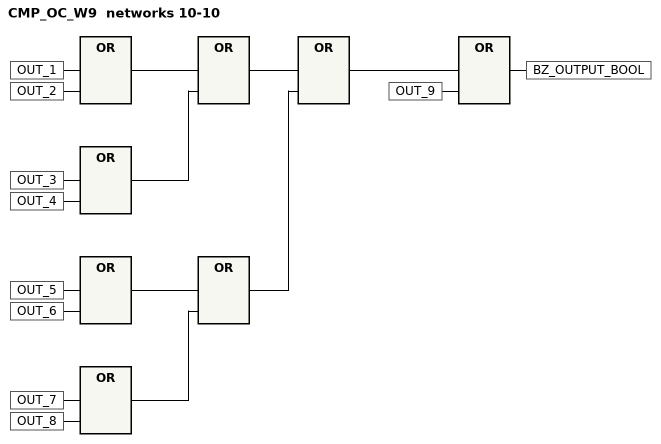
[picture p24: CMP_OC_W9 (FBD) networks 10-10]
_FBD_ (* Function Block Diagram *)
NETWORK 1
	OR(LT(WORD_1, 0), GT(WORD_1, 0)) => OUT_1
NETWORK 2
	OR(LT(WORD_2, 0), GT(WORD_2, 0)) => OUT_2
NETWORK 3
	OR(LT(WORD_3, 0), GT(WORD_3, 0)) => OUT_3
NETWORK 4
	OR(LT(WORD_4, 0), GT(WORD_4, 0)) => OUT_4
NETWORK 5
	OR(LT(WORD_5, 0), GT(WORD_5, 0)) => OUT_5
NETWORK 6
	OR(LT(WORD_6, 0), GT(WORD_6, 0)) => OUT_6
NETWORK 7
	OR(LT(WORD_7, 0), GT(WORD_7, 0)) => OUT_7
NETWORK 8
	OR(LT(WORD_8, 0), GT(WORD_8, 0)) => OUT_8
NETWORK 9
	OR(LT(WORD_9, 0), GT(WORD_9, 0)) => OUT_9
NETWORK 10
	OR(OR(OR(OR(OUT_1, OUT_2), OR(OUT_3, OUT_4)), OR(OR(OUT_5, OUT_6), OR(OUT_7, OUT_8))), OUT_9) => BZ_OUTPUT_BOOL
_END_FBD_
(* the same logic as Structured Text *)
(* Network 1 *)
OUT_1 := (WORD_1 < 0) OR (WORD_1 > 0);
(* Network 2 *)
OUT_2 := (WORD_2 < 0) OR (WORD_2 > 0);
(* Network 3 *)
OUT_3 := (WORD_3 < 0) OR (WORD_3 > 0);
(* Network 4 *)
OUT_4 := (WORD_4 < 0) OR (WORD_4 > 0);
(* Network 5 *)
OUT_5 := (WORD_5 < 0) OR (WORD_5 > 0);
(* Network 6 *)
OUT_6 := (WORD_6 < 0) OR (WORD_6 > 0);
(* Network 7 *)
OUT_7 := (WORD_7 < 0) OR (WORD_7 > 0);
(* Network 8 *)
OUT_8 := (WORD_8 < 0) OR (WORD_8 > 0);
(* Network 9 *)
OUT_9 := (WORD_9 < 0) OR (WORD_9 > 0);
(* Network 10 *)
BZ_OUTPUT_BOOL := (((OUT_1 OR OUT_2) OR (OUT_3 OR OUT_4)) OR ((OUT_5 OR OUT_6) OR (OUT_7 OR OUT_8))) OR OUT_9;
END_FUNCTION_BLOCK

(* POU DOWN_COUNT_TIMER, LD *)
FUNCTIONBLOCK DOWN_COUNT_TIMER
VAR_INPUT
	BOOL_SIGNAL_IN: BOOL;
	BOOL_TIMER_RST: BOOL;
	INT_AUTO_RST: INT;
	INT_SV_SEC: INT;
END_VAR
VAR_OUTPUT
	SIGNAL_BOOL: BOOL;
	PV_SEC_INT: INT;
END_VAR
VAR
	DF_1: R_TRIG;
	DF_2: R_TRIG;
	M1: BOOL;
	M2: BOOL;

	T100: TON;
	T101: TON;
	M100: BOOL;
	M101: BOOL;
	M200: BOOL;

	M110: BOOL;
	M300: BOOL;
END_VAR
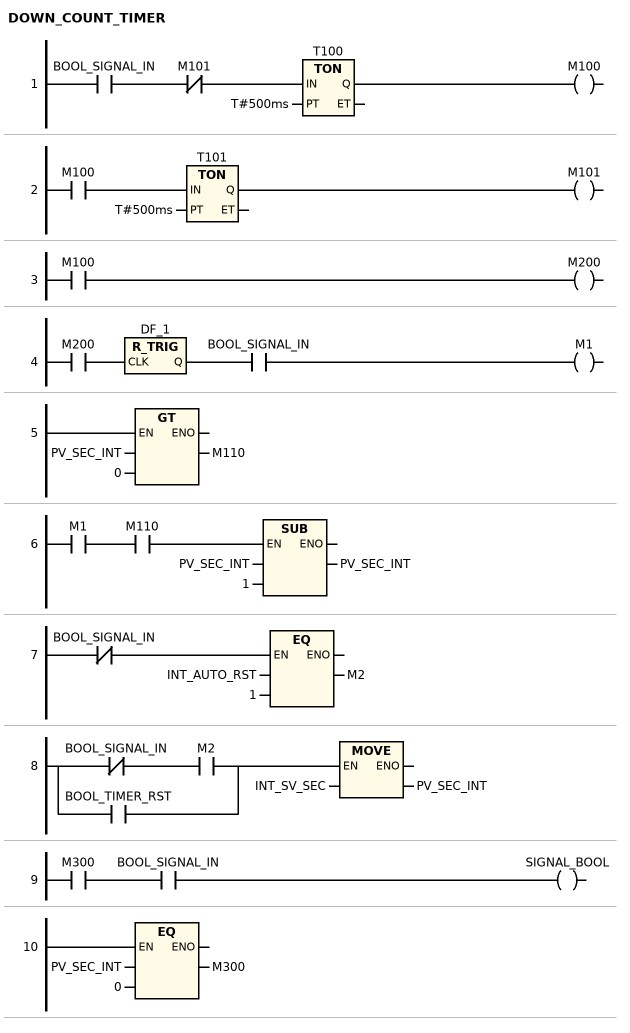
_LD_ (* Ladder Diagram *)
NETWORK 1
	[BOOL_SIGNAL_IN] - [/M101] - T100:TON(IN: *, PT: T#500ms) --- (M100)
NETWORK 2
	[M100] - T101:TON(IN: *, PT: T#500ms) --- (M101)
NETWORK 3
	[M100] --- (M200)
NETWORK 4
	[M200] - DF_1:R_TRIG(CLK: *) - [BOOL_SIGNAL_IN] --- (M1)
NETWORK 5
	*
		EN --- GT(PV_SEC_INT, 0) => M110
NETWORK 6
	[M1] - [M110]
		EN --- SUB(PV_SEC_INT, 1) => PV_SEC_INT
NETWORK 7
	[/BOOL_SIGNAL_IN]
		EN --- EQ(INT_AUTO_RST, 1) => M2
NETWORK 8
	{ [/BOOL_SIGNAL_IN] - [M2] | [BOOL_TIMER_RST] }
		EN --- MOVE(INT_SV_SEC) => PV_SEC_INT
NETWORK 9
	[M300] - [BOOL_SIGNAL_IN] --- (SIGNAL_BOOL)
NETWORK 10
	*
		EN --- EQ(PV_SEC_INT, 0) => M300
_END_LD_
(* the same logic as Structured Text *)
(* Network 1 *)
T100(IN := BOOL_SIGNAL_IN AND NOT M101, PT := T#500ms);
M100 := T100.Q;
(* Network 2 *)
T101(IN := M100, PT := T#500ms);
M101 := T101.Q;
(* Network 3 *)
M200 := M100;
(* Network 4 *)
DF_1(CLK := M200);
M1 := DF_1.Q AND BOOL_SIGNAL_IN;
(* Network 5 *)
M110 := PV_SEC_INT > 0;
(* Network 6 *)
IF M1 AND M110 THEN
	PV_SEC_INT := PV_SEC_INT - 1;
END_IF;
(* Network 7 *)
IF NOT BOOL_SIGNAL_IN THEN
	M2 := INT_AUTO_RST = 1;
END_IF;
(* Network 8 *)
IF NOT BOOL_SIGNAL_IN AND M2 OR BOOL_TIMER_RST THEN
	PV_SEC_INT := INT_SV_SEC;
END_IF;
(* Network 9 *)
SIGNAL_BOOL := M300 AND BOOL_SIGNAL_IN;
(* Network 10 *)
M300 := PV_SEC_INT = 0;
END_FUNCTION_BLOCK

(* POU CLOCK_PLS, LD *)
FUNCTION_BLOCK CLOCK_PLS
VAR_INPUT
	INT_TIME_ms : INT;

END_VAR
VAR_OUTPUT
	CLOCK_PLS_BOOL: BOOL;
END_VAR
VAR
	T0: TON;
	T1: TON;
	M0: BOOL;
	M1: BOOL;
	D0: TIME;
	D1: TIME;
END_VAR
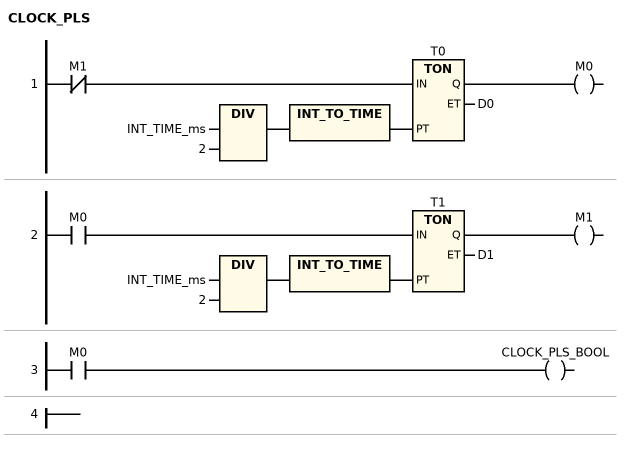
_LD_ (* Ladder Diagram *)
NETWORK 1
	[/M1] - T0:TON(IN: *, PT: INT_TO_TIME(DIV(INT_TIME_ms, 2)), ET => D0) --- (M0)
NETWORK 2
	[M0] - T1:TON(IN: *, PT: INT_TO_TIME(DIV(INT_TIME_ms, 2)), ET => D1) --- (M1)
NETWORK 3
	[M0] --- (CLOCK_PLS_BOOL)
NETWORK 4
	*
_END_LD_
(* the same logic as Structured Text *)
(* Network 1 *)
T0(IN := NOT M1, PT := INT_TO_TIME(INT_TIME_ms / 2));
D0 := T0.ET;
M0 := T0.Q;
(* Network 2 *)
T1(IN := M0, PT := INT_TO_TIME(INT_TIME_ms / 2));
D1 := T1.ET;
M1 := T1.Q;
(* Network 3 *)
CLOCK_PLS_BOOL := M0;
(* Network 4 *)
END_FUNCTION_BLOCK

(* POU EQ_GT, LD *)
FUNCTION_BLOCK EQ_GT
VAR_INPUT
	INT_SOURCE_A: INT;
	INT_SOURCE_B: INT;
END_VAR
VAR_OUTPUT
	SIGNAL_BOOL: BOOL;
END_VAR
VAR
	M0: BOOL;
	M1: BOOL;
END_VAR
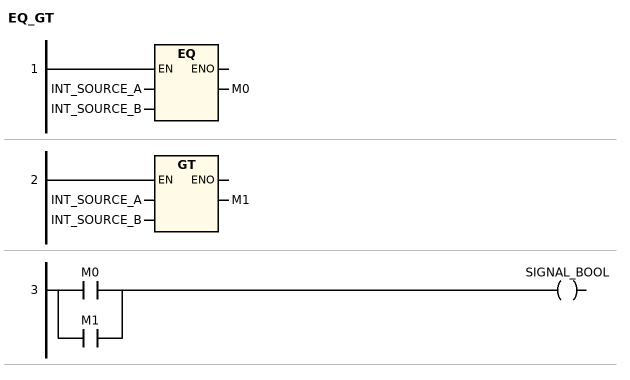
_LD_ (* Ladder Diagram *)
NETWORK 1
	*
		EN --- EQ(INT_SOURCE_A, INT_SOURCE_B) => M0
NETWORK 2
	*
		EN --- GT(INT_SOURCE_A, INT_SOURCE_B) => M1
NETWORK 3
	{ [M0] | [M1] } --- (SIGNAL_BOOL)
_END_LD_
(* the same logic as Structured Text *)
(* Network 1 *)
M0 := INT_SOURCE_A = INT_SOURCE_B;
(* Network 2 *)
M1 := INT_SOURCE_A > INT_SOURCE_B;
(* Network 3 *)
SIGNAL_BOOL := M0 OR M1;
END_FUNCTION_BLOCK

(* POU EQ_LT, LD *)
FUNCTION_BLOCK EQ_LT
VAR_INPUT
	INT_SOURCE_A:INT;
	INT_SOURCE_B:INT;
END_VAR
VAR_OUTPUT
	SIGNAL_BOOL:BOOL;
END_VAR
VAR
	M0: BOOL;
	M1: BOOL;
END_VAR
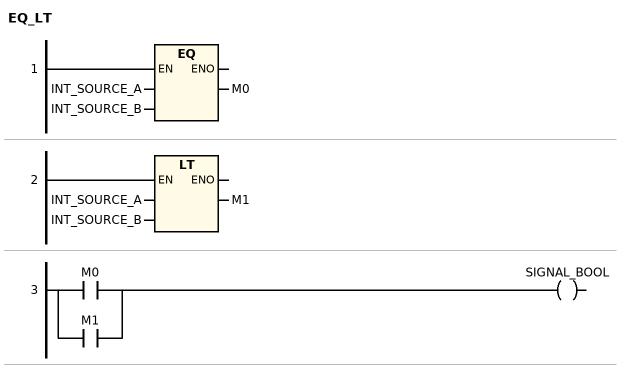
_LD_ (* Ladder Diagram *)
NETWORK 1
	*
		EN --- EQ(INT_SOURCE_A, INT_SOURCE_B) => M0
NETWORK 2
	*
		EN --- LT(INT_SOURCE_A, INT_SOURCE_B) => M1
NETWORK 3
	{ [M0] | [M1] } --- (SIGNAL_BOOL)
_END_LD_
(* the same logic as Structured Text *)
(* Network 1 *)
M0 := INT_SOURCE_A = INT_SOURCE_B;
(* Network 2 *)
M1 := INT_SOURCE_A < INT_SOURCE_B;
(* Network 3 *)
SIGNAL_BOOL := M0 OR M1;
END_FUNCTION_BLOCK

(* POU LT_GT, LD *)
FUNCTION_BLOCK LT_GT
VAR_INPUT
	INT_SOURCE_A: INT;
	INT_SOURCE_B: INT;
END_VAR
VAR_OUTPUT
	SIGNAL_BOOL: BOOL;
END_VAR
VAR
	M0: BOOL;
	M1: BOOL;
END_VAR
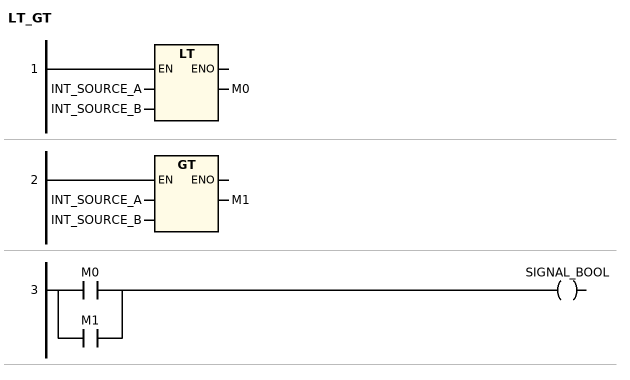
_LD_ (* Ladder Diagram *)
NETWORK 1
	*
		EN --- LT(INT_SOURCE_A, INT_SOURCE_B) => M0
NETWORK 2
	*
		EN --- GT(INT_SOURCE_A, INT_SOURCE_B) => M1
NETWORK 3
	{ [M0] | [M1] } --- (SIGNAL_BOOL)
_END_LD_
(* the same logic as Structured Text *)
(* Network 1 *)
M0 := INT_SOURCE_A < INT_SOURCE_B;
(* Network 2 *)
M1 := INT_SOURCE_A > INT_SOURCE_B;
(* Network 3 *)
SIGNAL_BOOL := M0 OR M1;
END_FUNCTION_BLOCK

(* POU TIMER_ALARM, LD *)
FUNCTION_BLOCK TIMER_ALARM
VAR_INPUT
	BOOL_SIGNAL_IN: BOOL;
	BOOL_ALMRST_PB: BOOL;
	BOOL_BZRST_PB: BOOL;
	INT_PV: INT;

END_VAR

VAR_OUTPUT
	ALM_MSG_BOOL: BOOL;
	BZ_OUT_BOOL: BOOL;
	EV_INT: INT;
END_VAR

VAR
	T1: TON;
	M0: BOOL;
	M1: BOOL;
	D200: TIME;
	D202: INT;
END_VAR
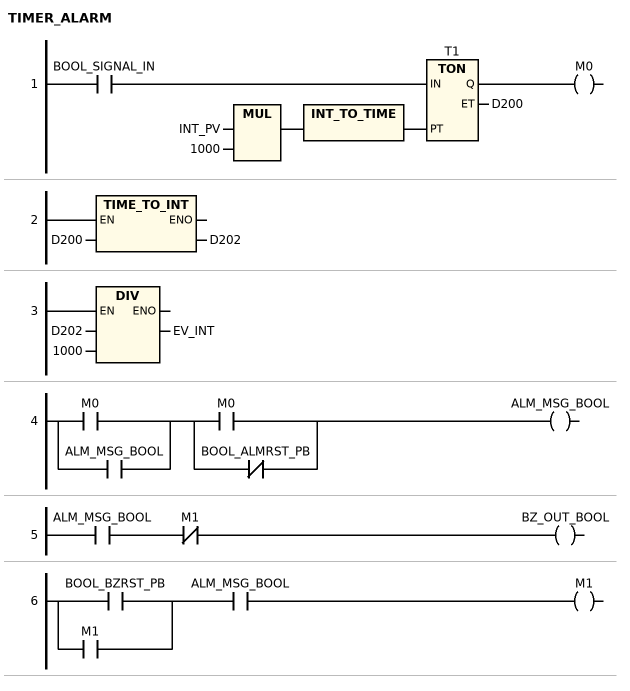
_LD_ (* Ladder Diagram *)
NETWORK 1
	[BOOL_SIGNAL_IN] - T1:TON(IN: *, PT: INT_TO_TIME(MUL(INT_PV, 1000)), ET => D200) --- (M0)
NETWORK 2
	*
		EN --- TIME_TO_INT(D200) => D202
NETWORK 3
	*
		EN --- DIV(D202, 1000) => EV_INT
NETWORK 4
	{ [M0] | [ALM_MSG_BOOL] } - { [M0] | [/BOOL_ALMRST_PB] } --- (ALM_MSG_BOOL)
NETWORK 5
	[ALM_MSG_BOOL] - [/M1] --- (BZ_OUT_BOOL)
NETWORK 6
	{ [BOOL_BZRST_PB] | [M1] } - [ALM_MSG_BOOL] --- (M1)
_END_LD_
(* the same logic as Structured Text *)
(* Network 1 *)
T1(IN := BOOL_SIGNAL_IN, PT := INT_TO_TIME(INT_PV * 1000));
D200 := T1.ET;
M0 := T1.Q;
(* Network 2 *)
D202 := TIME_TO_INT(D200);
(* Network 3 *)
EV_INT := D202 / 1000;
(* Network 4 *)
ALM_MSG_BOOL := (M0 OR ALM_MSG_BOOL) AND (M0 OR NOT BOOL_ALMRST_PB);
(* Network 5 *)
BZ_OUT_BOOL := ALM_MSG_BOOL AND NOT M1;
(* Network 6 *)
M1 := (BOOL_BZRST_PB OR M1) AND ALM_MSG_BOOL;
END_FUNCTION_BLOCK
